Staubli VAL3: onF2Event.pgx

program onF2Event()
  local string l_sItem
  local string l_sPage
begin
  // look if the bButton is enable
  if bButton[1]
    //
    //
    l_sPage="trajectory/page_trajectory"
    call loadPage(l_sPage,l_sItem)
    logMsg("[KERNEL] INTERFACE:PAGE Home Page")
  endIf
end
